ABB RAPID module: MainModule.mod

MODULE MainModule
  !*********************************************************
  !Subject: Tcp definition 4 way
  !Robot Type: IRB2600
  !Author:   jun byouang lee
  !Revision: 2020-05-31
  !*********************************************************
  CONST robtarget p10:=[[850,-250,750],[0.000039112,0.000013788,1,-0.000000552],[-1,-1,0,1],[9E+09,9E+09,9E+09,9E+09,9E+09,9E+09]];
  CONST robtarget p20:=[[1000,-250,700],[0.000039281,0.000013614,1,-0.000000204],[-1,-1,0,1],[9E+09,9E+09,9E+09,9E+09,9E+09,9E+09]];
  CONST robtarget p30:=[[1000,50,700],[0.000040124,0.000014118,1,0.000000242],[0,0,-1,1],[9E+09,9E+09,9E+09,9E+09,9E+09,9E+09]];
  CONST robtarget p40:=[[1100,150,700],[0.000042484,0.000013371,1,0.00000093],[0,0,-1,1],[9E+09,9E+09,9E+09,9E+09,9E+09,9E+09]];
  CONST robtarget p50:=[[1000,250,700],[0.000040967,0.000013858,1,0.000000464],[0,0,-1,1],[9E+09,9E+09,9E+09,9E+09,9E+09,9E+09]];
  CONST robtarget pHome:=[[700.00,0.00,950.00],[0.707107,-3.44283E-9,0.707107,-3.44283E-9],[0,0,-1,0],[9E+9,9E+9,9E+9,9E+9,9E+9,9E+9]];

  PROC main()
    MoveJ pHome, v300, fine, tool0;
    !test
  ENDPROC
ENDMODULE
